FUNCTION_BLOCK PUBLIC FB_CANControl IMPLEMENTS ITF_CANControl
VAR_INPUT
END_VAR
VAR_OUTPUT
END_VAR
VAR
	rxQueue AT%I* : ST_TxRxQueue;
	txQueue AT%Q* : ST_TxRxQueue;
	i : INT;
	messageRecieved : ST_TxRxMessage;
END_VAR

IF rxQueue.rxCounter <> txQueue.rxCounter THEN
	//if we have recieved a message rxCounter is incremented by interface
	M_GetMessage();
END_IF

METHOD PUBLIC M_GetMessage : BOOL
VAR_INPUT
END_VAR
FOR i := 0 TO rxQueue.noOfMessages DO
	messageRecieved := rxQueue.messages[i];
END_FOR
txQueue.rxCounter := rxQueue.rxCounter;
END_METHOD

METHOD PUBLIC M_PushMessage : BOOL
VAR_INPUT
	messageSend : ST_TxRxMessage;
END_VAR
IF txQueue.txCounter = rxQueue.TxCounter THEN
	FOR i:=0 TO 1 DO
		txQueue.messages[i] := messageSend;
	End_for
	txQueue.noOfMessages := 1;
	txQueue.TxCounter := rxQueue.TxCounter + 1;
END_IF
END_METHOD

END_FUNCTION_BLOCK

(* stored: Version 1.1.0.1, ProductVersion 3.1.4024.11
   POU FB_CANControl: Id {01544bbb-d8cd-408f-acf6-6133198b589f}, SpecialFunc None
   Method M_GetMessage: Id {98350e53-ad4f-48fd-8cf0-20480dae082c}
   Method M_PushMessage: Id {16f7dc02-3cbc-4c81-ab5b-858e74097005} *)
